(* Logix 5000 project; controller MetsoFilter vendor 1 type 14 code 106 rev 32.11; software revision 32.00; part 2 of 4 *)
(* tags used below, declared in another part *)
   AlarmReset : BOOL;   // Alarm Rest Relay
   ALM_AirAndWaterOK_T : TIMER;   // Air and Water OK, Enable Air & Water Valves Alarms
   ALM_W1 : DINT;   // Alarms to HMI, Word #1
   ALM_W2 : DINT;   // Alarms to HMI, Word #2
   AS_AirDry : BOOL;   // Auto Sequence, Air Dry
   AS_ClothFlush : BOOL;   // Auto Sequence Flush out Cloth
   AS_ClothFlush_T : TIMER;   // Auto Sequence Flush out Cloth Timer
   AS_ClothVibWash : BOOL;   // Auto Sequence Vibrate & Wash Cloth
   AS_ClothVibWash_T : TIMER;   // Auto Sequence Vibrate & Wash Cloth Timer
   AS_Done : BOOL;   // Automatic Sequence Done, Reset Sequence for Next Run
   AS_Drain : BOOL;   // Auto Sequence, Drain
   AS_FeedFilter : BOOL;   // Auto Sequence, Feed Filter
   AS_HighEmptyWeight : BOOL;   // Auto Sequence, High Empty Weight, Manually Shake filter
   AS_HighPressClose : BOOL;   // Auto Sequence, Close Press at High Pressure
   AS_LowFeedWeight : BOOL;   // Auto Sequence, Low Feed Weight, Enable Retry
   AS_LowPressClose : BOOL;   // Auto Sequence, Close Press at Low Pressure
   AS_MembComp : BOOL;   // Auto Sequence, Membrane Compress
   AS_TopBlowAir1 : BOOL;   // Auto Sequence, Top Blow Air #1
   AS_TopBlowAir2 : BOOL;   // Auto Sequence, Top Blow Air #2
   AS_TopBlowWat : BOOL;   // Automatic Sequence, Top Blow & Water
   AS_VibrateCloth : BOOL;   // Auto Sequence Vibrate Cloth
   AS_VibrateCloth_T : TIMER;   // Auto Sequence Vibrate Cloth Timer
   AS_Wait : BOOL;   // Auto Sequence Wait
   AS_Wait_T : TIMER;   // Auto Sequence Wait Timer
   At_Parked_Pos_T : TIMER;   // Press At Parked (Closed) Postion Timer
   Auto_ON : BOOL;   // Auto On Mode
   Auto_Run : BOOL;   // Run the Next Step of the Auto Sequence
   AutoSeqStarted : BOOL;   // Auto Sequence Started
   DD_PressPressure : REAL;   // Press Pressure Data Display
   DD_PressWeight : DINT;   // Press Weight from Analog Input Data Display
   DE_ClothVibWash : DINT;   // Settings Screen, Cloth Vibrate and Wash Time Data Entry (Seconds)
   DE_ClothWash : DINT;   // Settings Screen, Cloth Wash Time Data Entry (Seconds)
   DE_DelayedStart : DINT;   // Settings Screen, Delay Start Wait Time Data Entry (Seconds)
   DryAirSwitch : BOOL;   // Drying Air OK Switch
   Goto_Neutral_T : TIMER;   // Manual / Auto Open (Goto Neutral) Press On Plus Time
   Goto_Park_T : TIMER;   // Go to Park On Plus Time
   Goto_Press_T : TIMER;   // Go to Press Position Output On Plus Time
   GS3 : BOOL;   // Press At Park Position Prox Switch
   GS4 : BOOL;   // Press At Neutral Position Prox Switch
   GS8 : BOOL;   // Press At Press Position Prox Switch
   GSC11 : BOOL;   // Upper Hatch is Closed Proximity Switch
   GSC9 : BOOL;   // Lower Hatch is Closed Proximity Switch
   GSO10 : BOOL;   // Lower Hatch is Open Proximity Switch
   GSO12 : BOOL;   // Upper Hatch is Open Proximity Switch
   H4a : BOOL;   // Hydraulic Valve, Raise (Open) Lower Hatch
   H4a_On_T : TIMER;   // Hydraulic Valve, Raise (Open) Lower Hatch On Plus Time
   H4b : BOOL;   // Hydraulic Valve, Lower (Close) Lower Hatch
   H4b_On_T : TIMER;   // Hydraulic Valve, Lower (Close) Lower Hatch On Plus Time
   H5a : BOOL;   // Hydraulic Valve, Raise (Open) Upper Hatch
   H5a_On_T : TIMER;   // Hydraulic Valve, Raise (Open) Upper Hatch On Plus Time
   H5b : BOOL;   // Hydraulic Valve, Lower (Close) Upper Hatch
   H5b_On_T : TIMER;   // Hydraulic Valve, Lower (Close) Upper Hatch On Plus Time
   HPP_Run_T : TIMER;   // High Pressure Pump Run Timer
   LPP_Run_T : TIMER;   // Low Pressure Pump Run Timer
   M_HPP_Run : BOOL;   // High Pressure Pump Run Output Bit
   M_HPP_Running : BOOL;   // High Pressure Pump is Running
   M_LPP_Run : BOOL;   // Low Pressure Pump Run Output Bit
   M_LPP_Running : BOOL;   // Low Pressure Pump is Running
   MAN_ClosePress : BOOL;   // Manual Close Press to Park Position
   Manual_ON : BOOL;   // Manual On Mode
   MAS_CloseHatch : BOOL;   // Manual / Auto Close Hatch
   MAS_HatchesClosed_T : TIMER;   // Manual / Auto Hatchs are Closed + Time
   MAS_OpenHatch : BOOL;   // Manual / Auto Open Hatch
   MAS_OpenPress : BOOL;   // Manual / Auto Open (Goto Neutral) Press
   MSG_Activity : DINT;   // Activity Message display at left side of the HMI Screens.
   MSG_CloseHatch : BOOL;   // Show Closing Hatches in Sequence & Activity messages latch
   MSG_Main : DINT;   // Main Message at center of screen,
   MSG_MainTemp : DINT;   // Main Message at center of screen, Temporary Holding Register
   MSG_OpenHatch : BOOL;   // Show Opeining Hatch in SEquence & Activity messages latch
   MSG_OpenPress : BOOL;   // Show Opeining Press in Sequence & Activity messages latch
   MSG_SeqTemp : DINT;   // Sequence & Activity Message displays at left side of the HMI Screens, Temp hold
   MSG_Sequence : DINT;   // Sequence Message display at left side of the HMI Screens.
   NumberOfAlarms : DINT;   // Number of Active Alarms
   PressPressure_OOR_T : TIMER;   // Press Pressure Sensor Out Of Range Plus Time
   PressWeight_OOR_T : TIMER;   // Press Weight Out Of Range Timer
   SlurrySystemSwitch : BOOL;   // Slurry System OK Switch
   V10_GSC : BOOL;   // Valve #10, Membrane Drain, Closed Input
   V10_Off_T : TIMER;   // Valve #10, Membrane Drain, Ouput Bit Off Plus Time, Valve shoud be Open
   V10_On_T : TIMER;   // Valve #10, Membrane Drain, Ouput Bit On Plus Time, Valve shoud be Closed
   V1_GSC : BOOL;   // Valve #1, Slurry Supply, Closed Input
   V1_GSO : BOOL;   // Valve #1, Slurry Supply, Open Input
   V1_Off_T : TIMER;   // Valve #1, Slurry Supply, Open Output Bit Off Plus Time
   V1_On_T : TIMER;   // Valve #1, Slurry Supply, Open Output Bit On Plus Time
   V3_GSC : BOOL;   // Valve #3, Filtrate, Closed Input
   V3_GSO : BOOL;   // Valve #3, Filtrate, Open Input
   V3_Off_T : TIMER;   // Valve #3, Filtrate, Open Output Bit Off Plus time
   V3_On_T : TIMER;   // Valve #3, Filtrate, Open Output Bit On Plus time
   V4_GSC : BOOL;   // Valve #4, Slurry Return, Closed Input
   V4_GSO : BOOL;   // Valve #4, Slurry Return, Open Input
   V4_Off_T : TIMER;   // Valve #4, Slurry Return, Open Output Bit Off Plus Time
   V4_On_T : TIMER;   // Valve #4, Slurry Return, Open Output Bit On Plus Time
   V5_GSC : BOOL;   // Valve #5, Drying Air, Closed Input
   V5_GSO : BOOL;   // Valve #5, Drying Air, Opened Input
   V5_Off_T : TIMER;   // Valve #5, Drying Air, Open Output Bit Off Plus Time
   V5_On_T : TIMER;   // Valve #5, Drying Air, Open Output Bit On Plus Time
   V6_GSC : BOOL;   // Valve #6, Top Blow Air, Closed Input
   V6_GSO : BOOL;   // Valve #6, Top Blow Air, Opened Input
   V6_Off_T : TIMER;   // Valve #6, Top Blow Air, Open Output Bit On Plus Time
   V6_On_T : TIMER;   // Valve #6, Top Blow Air, Open Output Bit On Plus Time
   V7_GSC : BOOL;   // Valve #7, Membrane Air, Closed Input
   V7_GSO : BOOL;   // Valve #7, Membrane Air, Opened Input
   V7_Off_T : TIMER;   // Valve #7, Membrane Air, Open Output Bit Off Plus Time
   V7_On_T : TIMER;   // Valve #7, Membrane Air, Open Output Bit On Plus time
   V8_GSC : BOOL;   // Valve #8, Top Blow Water, Closed Input
   V8_GSO : BOOL;   // Valve #8, Top Blow Water, Opened Input
   V8_Off_T : TIMER;   // Valve #8, Top Blow Water, Open Output Bit Off Plus Time
   V8_On_T : TIMER;   // Valve #8, Top Blow Water, Open Output Bit On Plus Time
   V9_GSC : BOOL;   // Valve #9, Wash Water, Closed Input
   V9_GSO : BOOL;   // Valve #9, Wash Water, Opened Input
   V9_Off_T : TIMER;   // Valve #9, Wash Water, Open Ouput Bit Off Plus Time
   V9_On_T : TIMER;   // Valve #9, Wash Water, Open Ouput Bit On Plus Time
   WashWaterSwitch : BOOL;   // Wash Water System OK Switch
   YV1 : BOOL;   // Valve #1, Slurry Supply, Open Output Bit
   YV10 : BOOL;   // Valve #10, Membrane Drain, Normally Open, Energize to Close, Output Bit
   YV3 : BOOL;   // Valve #3, Filtrate, Open Output Bit
   YV4 : BOOL;   // Valve #4, Slurry Return, Open Output Bit
   YV5 : BOOL;   // Valve #5, Drying Air, Open Output Bit
   YV6 : BOOL;   // Valve #6, Top Blow Air, Open Output Bit
   YV7 : BOOL;   // Valve #7, Membrane Air, Open Output Bit
   YV8 : BOOL;   // Valve #8, Top Blow Water, Open Output Bit
   YV9 : BOOL;   // Valve #9, Wash Water, Open Ouput Bit
(* MainProgram, continued *)

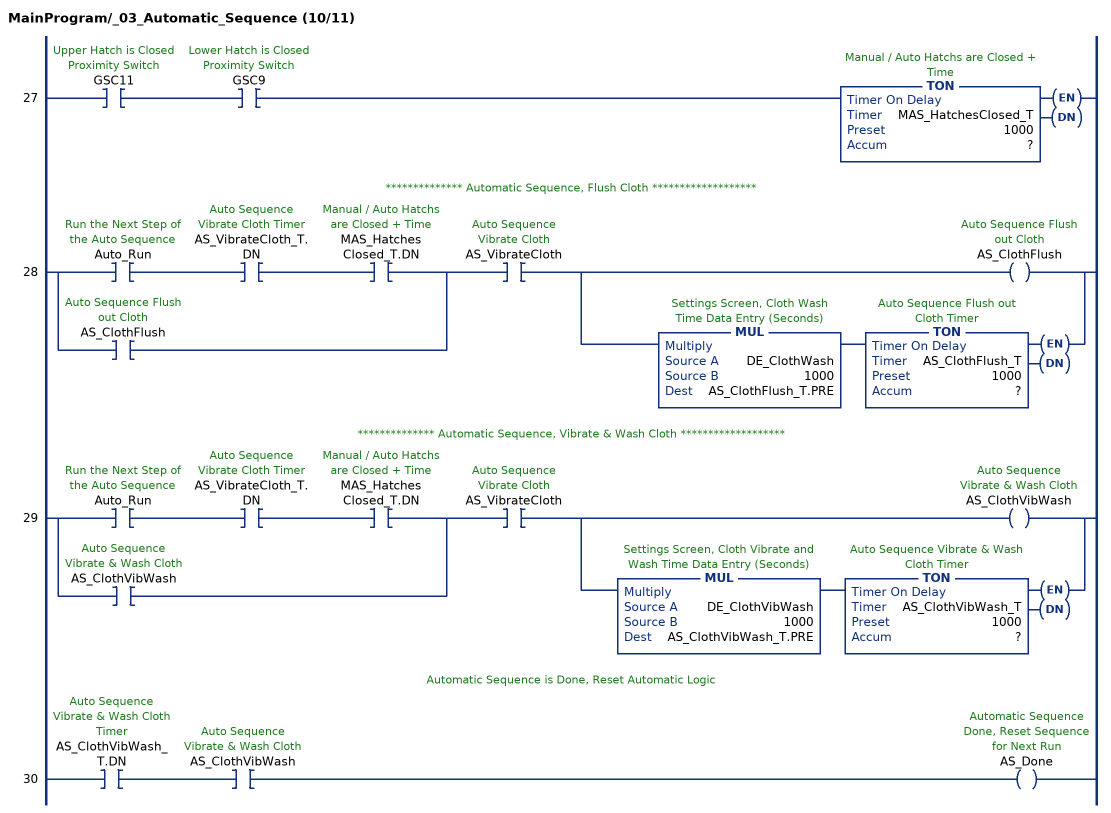
   [picture p24: MainProgram/_03_Automatic_Sequence rungs 27-30]
   27: XIC(GSC11)XIC(GSC9)TON(MAS_HatchesClosed_T,?,?);
   // ************** Automatic Sequence, Flush Cloth *******************
   28: [XIC(Auto_Run) XIC(AS_VibrateCloth_T.DN) XIC(MAS_HatchesClosed_T.DN) ,XIC(AS_ClothFlush) ]XIC(AS_VibrateCloth)[OTE(AS_ClothFlush) ,MUL(DE_ClothWash,1000,AS_ClothFlush_T.PRE) TON(AS_ClothFlush_T,?,?) ];
   // ************** Automatic Sequence, Vibrate & Wash Cloth *******************
   29: [XIC(Auto_Run) XIC(AS_VibrateCloth_T.DN) XIC(MAS_HatchesClosed_T.DN) ,XIC(AS_ClothVibWash) ]XIC(AS_VibrateCloth)[OTE(AS_ClothVibWash) ,MUL(DE_ClothVibWash,1000,AS_ClothVibWash_T.PRE) TON(AS_ClothVibWash_T,?,?) ];
   // Automatic Sequence is Done, Reset Automatic Logic
   30: XIC(AS_ClothVibWash_T.DN)XIC(AS_ClothVibWash)OTE(AS_Done);
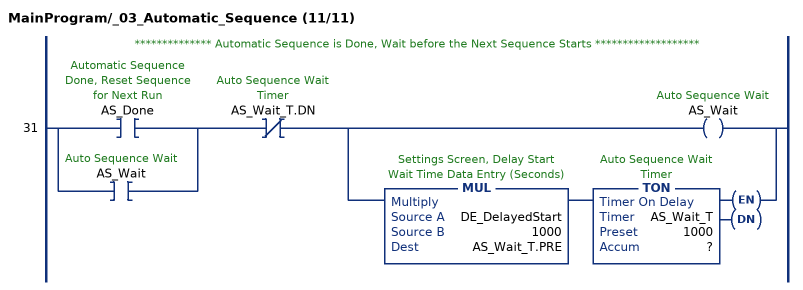
   // ************** Automatic Sequence is Done, Wait before the Next Sequence Starts *******************
   31: [XIC(AS_Done) ,XIC(AS_Wait) ]XIO(AS_Wait_T.DN)[OTE(AS_Wait) ,MUL(DE_DelayedStart,1000,AS_Wait_T.PRE) TON(AS_Wait_T,?,?) ];
END_ROUTINE

ROUTINE _04_HMI_MessageDisplays   (* ladder *)
// Message Displays on HMI Screens
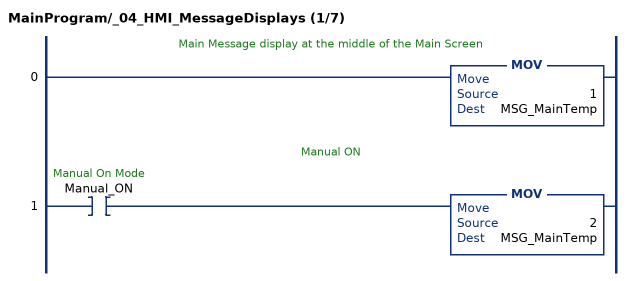
   // Main Message display at the middle of the Main Screen
   0: MOV(1,MSG_MainTemp);
   // Manual ON
   1: XIC(Manual_ON)MOV(2,MSG_MainTemp);
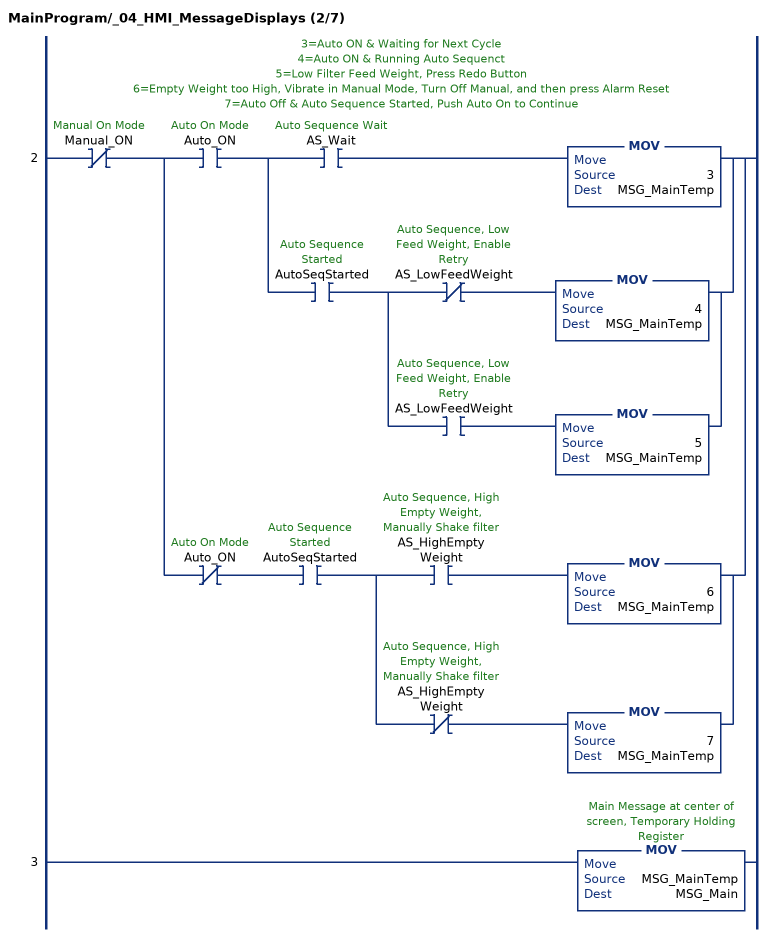
   // 3=Auto ON & Waiting for Next Cycle
   // 4=Auto ON & Running Auto Sequenct
   // 5=Low Filter Feed Weight, Press Redo Button
   // 6=Empty Weight too High, Vibrate in Manual Mode, Turn Off Manual, and then press Alarm Reset
   // 7=Auto Off & Auto Sequence Started, Push Auto On to Continue
   2: XIO(Manual_ON)[XIC(Auto_ON) [XIC(AS_Wait) MOV(3,MSG_MainTemp) ,XIC(AutoSeqStarted) [XIO(AS_LowFeedWeight) MOV(4,MSG_MainTemp) ,XIC(AS_LowFeedWeight) MOV(5,MSG_MainTemp) ] ] ,XIO(Auto_ON) XIC(AutoSeqStarted) [XIC(AS_HighEmptyWeight) MOV(6,MSG_MainTemp) ,XIO(AS_HighEmptyWeight) MOV(7,MSG_MainTemp) ] ];
   3: MOV(MSG_MainTemp,MSG_Main);
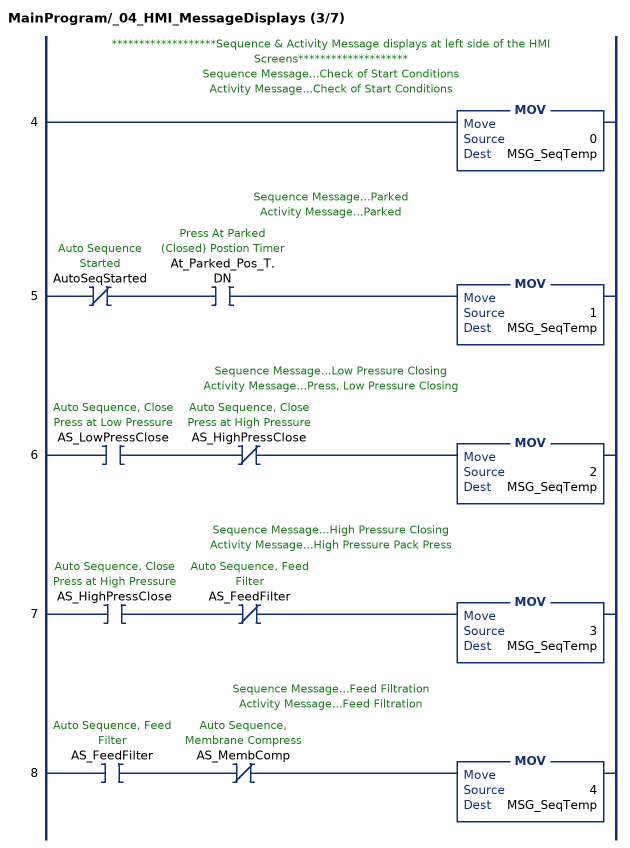
   // *******************Sequence & Activity Message displays at left side of the HMI Screens********************
   // Sequence Message...Check of Start Conditions
   // Activity Message...Check of Start Conditions
   4: MOV(0,MSG_SeqTemp);
   // Sequence Message...Parked
   // Activity Message...Parked
   5: XIO(AutoSeqStarted)XIC(At_Parked_Pos_T.DN)MOV(1,MSG_SeqTemp);
   // Sequence Message...Low Pressure Closing
   // Activity Message...Press, Low Pressure Closing
   6: XIC(AS_LowPressClose)XIO(AS_HighPressClose)MOV(2,MSG_SeqTemp);
   // Sequence Message...High Pressure Closing
   // Activity Message...High Pressure Pack Press
   7: XIC(AS_HighPressClose)XIO(AS_FeedFilter)MOV(3,MSG_SeqTemp);
   // Sequence Message...Feed Filtration
   // Activity Message...Feed Filtration
   8: XIC(AS_FeedFilter)XIO(AS_MembComp)MOV(4,MSG_SeqTemp);
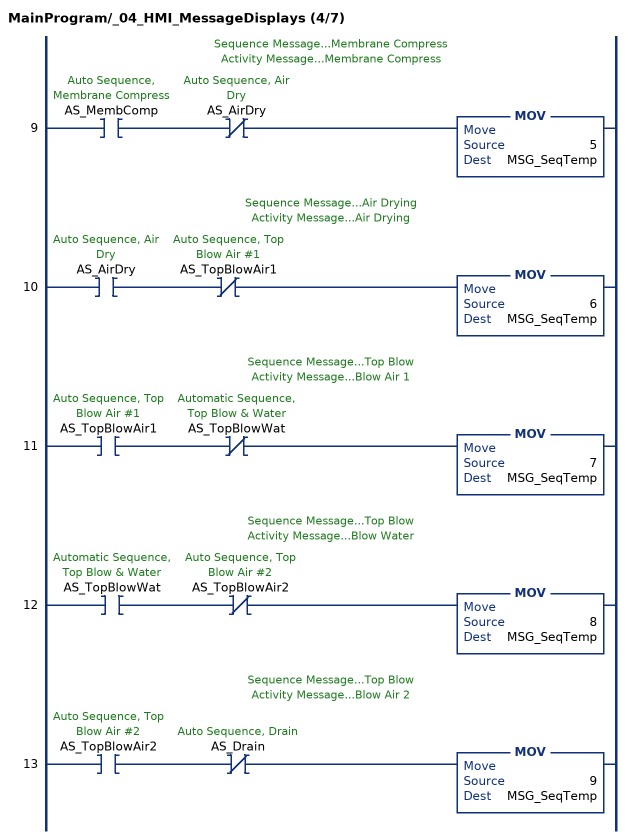
   // Sequence Message...Membrane Compress
   // Activity Message...Membrane Compress
   9: XIC(AS_MembComp)XIO(AS_AirDry)MOV(5,MSG_SeqTemp);
   // Sequence Message...Air Drying
   // Activity Message...Air Drying
   10: XIC(AS_AirDry)XIO(AS_TopBlowAir1)MOV(6,MSG_SeqTemp);
   // Sequence Message...Top Blow
   // Activity Message...Blow Air 1
   11: XIC(AS_TopBlowAir1)XIO(AS_TopBlowWat)MOV(7,MSG_SeqTemp);
   // Sequence Message...Top Blow
   // Activity Message...Blow Water
   12: XIC(AS_TopBlowWat)XIO(AS_TopBlowAir2)MOV(8,MSG_SeqTemp);
   // Sequence Message...Top Blow
   // Activity Message...Blow Air 2
   13: XIC(AS_TopBlowAir2)XIO(AS_Drain)MOV(9,MSG_SeqTemp);
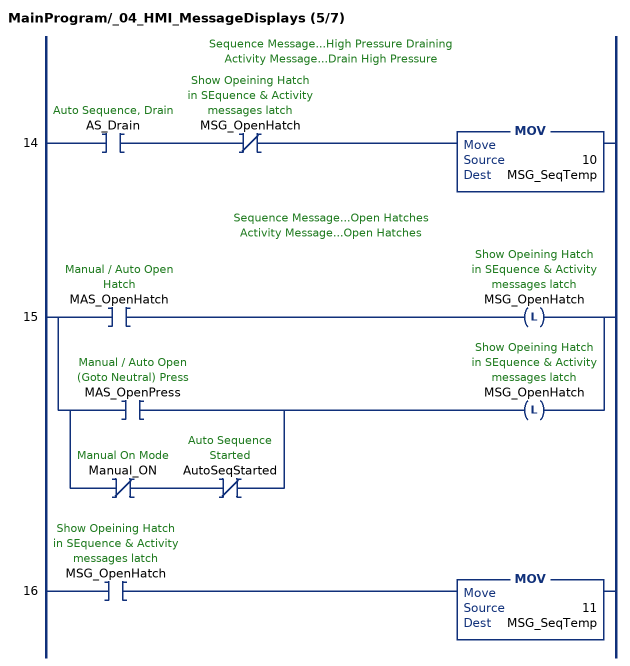
   // Sequence Message...High Pressure Draining
   // Activity Message...Drain High Pressure
   14: XIC(AS_Drain)XIO(MSG_OpenHatch)MOV(10,MSG_SeqTemp);
   // Sequence Message...Open Hatches
   // Activity Message...Open Hatches
   15: [XIC(MAS_OpenHatch) OTL(MSG_OpenHatch) ,[XIC(MAS_OpenPress) ,XIO(Manual_ON) XIO(AutoSeqStarted) ] OTL(MSG_OpenHatch) ];
   16: XIC(MSG_OpenHatch)MOV(11,MSG_SeqTemp);
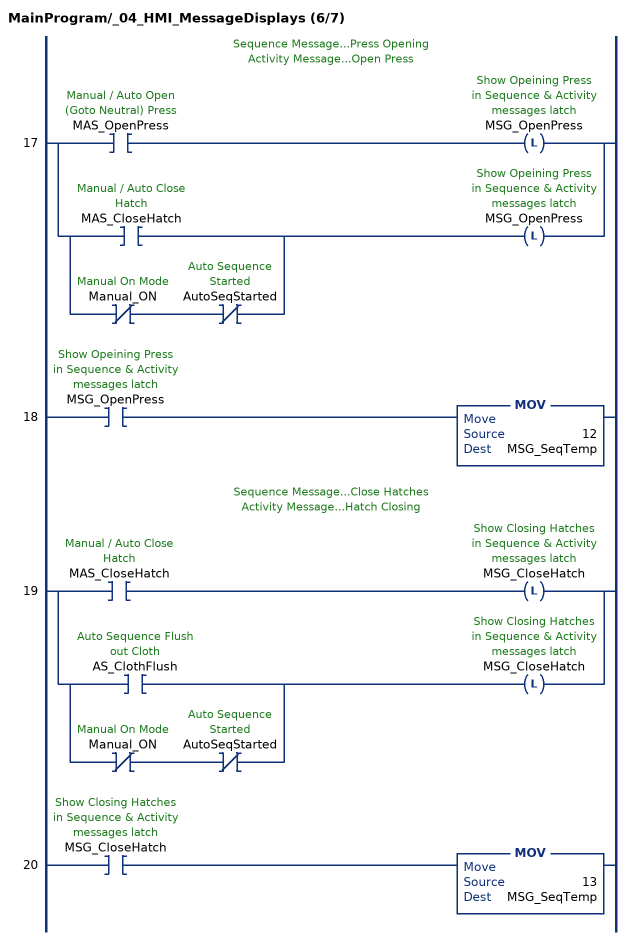
   // Sequence Message...Press Opening
   // Activity Message...Open Press
   17: [XIC(MAS_OpenPress) OTL(MSG_OpenPress) ,[XIC(MAS_CloseHatch) ,XIO(Manual_ON) XIO(AutoSeqStarted) ] OTL(MSG_OpenPress) ];
   18: XIC(MSG_OpenPress)MOV(12,MSG_SeqTemp);
   // Sequence Message...Close Hatches
   // Activity Message...Hatch Closing
   19: [XIC(MAS_CloseHatch) OTL(MSG_CloseHatch) ,[XIC(AS_ClothFlush) ,XIO(Manual_ON) XIO(AutoSeqStarted) ] OTL(MSG_CloseHatch) ];
   20: XIC(MSG_CloseHatch)MOV(13,MSG_SeqTemp);
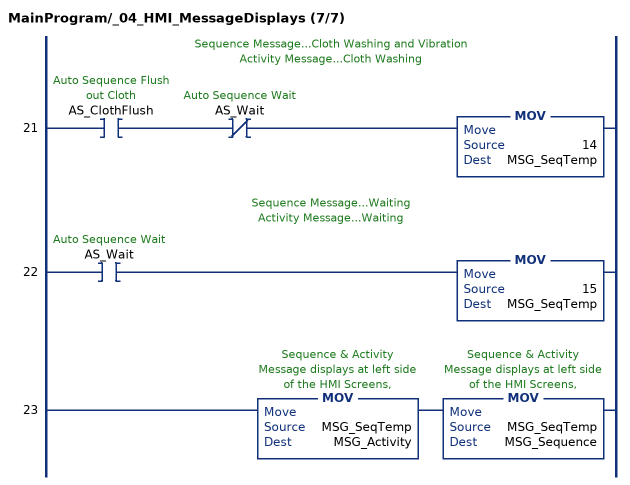
   // Sequence Message...Cloth Washing and Vibration
   // Activity Message...Cloth Washing
   21: XIC(AS_ClothFlush)XIO(AS_Wait)MOV(14,MSG_SeqTemp);
   // Sequence Message...Waiting
   // Activity Message...Waiting
   22: XIC(AS_Wait)MOV(15,MSG_SeqTemp);
   23: MOV(MSG_SeqTemp,MSG_Activity)MOV(MSG_SeqTemp,MSG_Sequence);
END_ROUTINE

ROUTINE _05_Alarms   (* ladder *)
// Alarms Logic
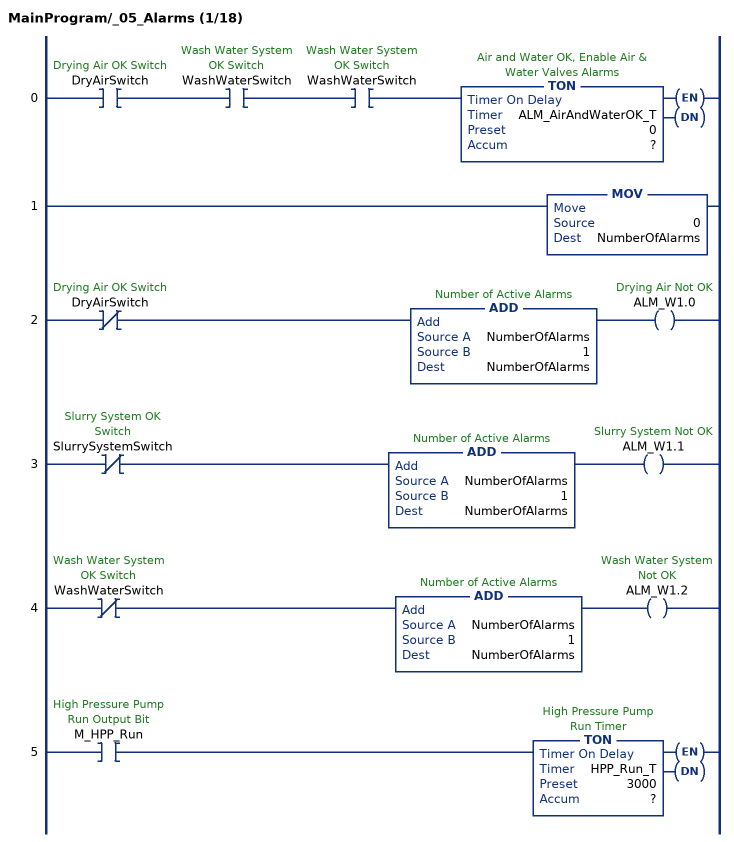
   0: XIC(DryAirSwitch)XIC(WashWaterSwitch)XIC(WashWaterSwitch)TON(ALM_AirAndWaterOK_T,?,?);
   1: MOV(0,NumberOfAlarms);
   2: XIO(DryAirSwitch)ADD(NumberOfAlarms,1,NumberOfAlarms)OTE(ALM_W1.0);
   3: XIO(SlurrySystemSwitch)ADD(NumberOfAlarms,1,NumberOfAlarms)OTE(ALM_W1.1);
   4: XIO(WashWaterSwitch)ADD(NumberOfAlarms,1,NumberOfAlarms)OTE(ALM_W1.2);
   5: XIC(M_HPP_Run)TON(HPP_Run_T,?,?);
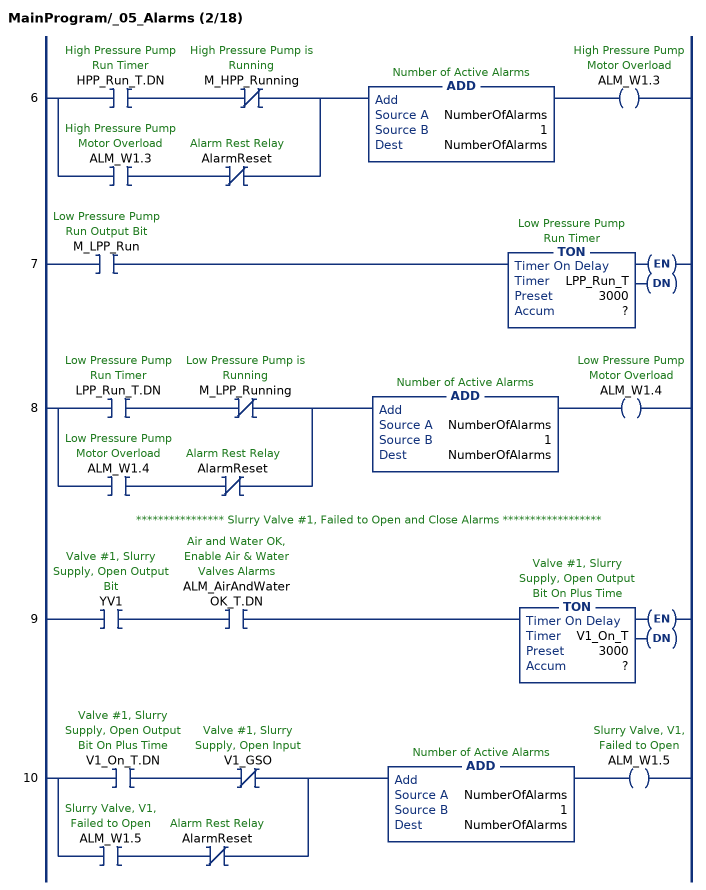
   6: [XIC(HPP_Run_T.DN) XIO(M_HPP_Running) ,XIC(ALM_W1.3) XIO(AlarmReset) ]ADD(NumberOfAlarms,1,NumberOfAlarms)OTE(ALM_W1.3);
   7: XIC(M_LPP_Run)TON(LPP_Run_T,?,?);
   8: [XIC(LPP_Run_T.DN) XIO(M_LPP_Running) ,XIC(ALM_W1.4) XIO(AlarmReset) ]ADD(NumberOfAlarms,1,NumberOfAlarms)OTE(ALM_W1.4);
   // **************** Slurry Valve #1, Failed to Open and Close Alarms ******************
   9: XIC(YV1)XIC(ALM_AirAndWaterOK_T.DN)TON(V1_On_T,?,?);
   10: [XIC(V1_On_T.DN) XIO(V1_GSO) ,XIC(ALM_W1.5) XIO(AlarmReset) ]ADD(NumberOfAlarms,1,NumberOfAlarms)OTE(ALM_W1.5);
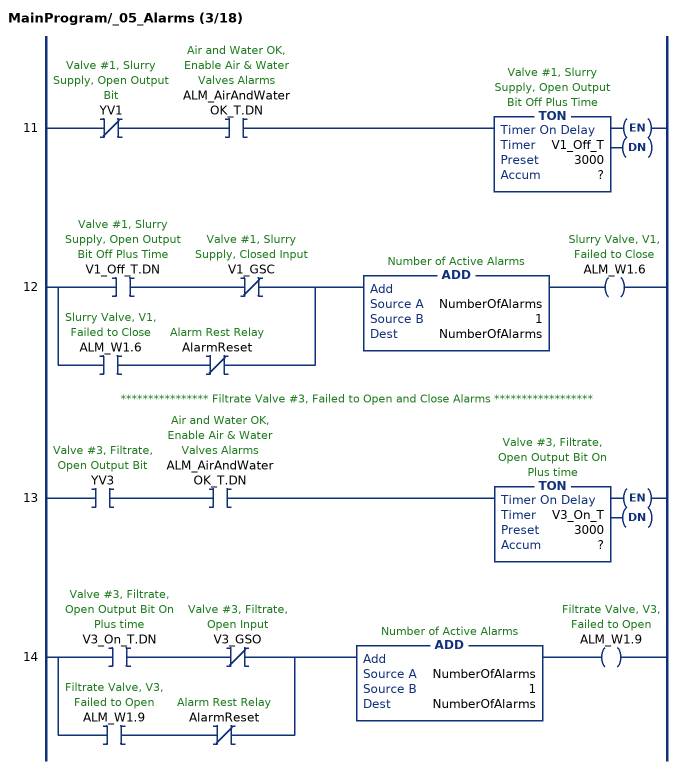
   11: XIO(YV1)XIC(ALM_AirAndWaterOK_T.DN)TON(V1_Off_T,?,?);
   12: [XIC(V1_Off_T.DN) XIO(V1_GSC) ,XIC(ALM_W1.6) XIO(AlarmReset) ]ADD(NumberOfAlarms,1,NumberOfAlarms)OTE(ALM_W1.6);
   // **************** Filtrate Valve #3, Failed to Open and Close Alarms ******************
   13: XIC(YV3)XIC(ALM_AirAndWaterOK_T.DN)TON(V3_On_T,?,?);
   14: [XIC(V3_On_T.DN) XIO(V3_GSO) ,XIC(ALM_W1.9) XIO(AlarmReset) ]ADD(NumberOfAlarms,1,NumberOfAlarms)OTE(ALM_W1.9);
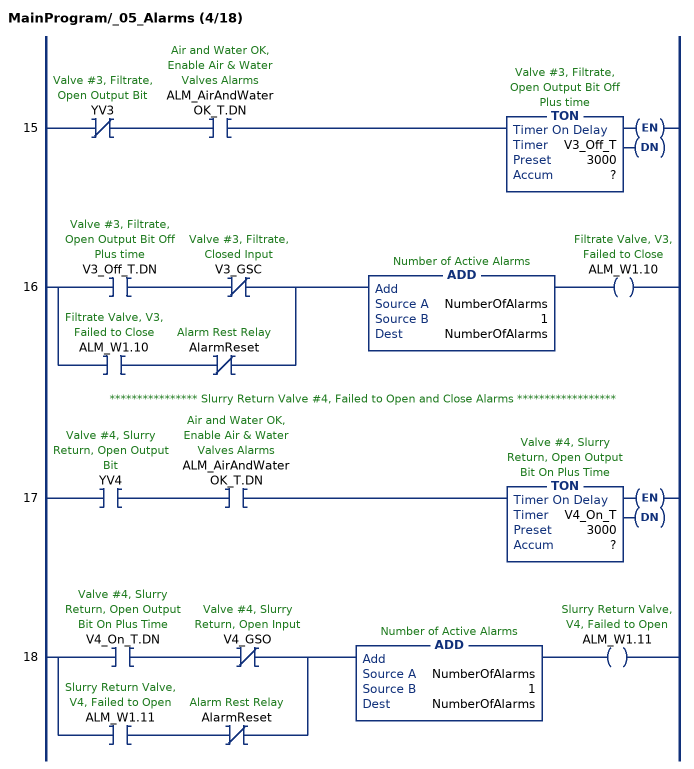
   15: XIO(YV3)XIC(ALM_AirAndWaterOK_T.DN)TON(V3_Off_T,?,?);
   16: [XIC(V3_Off_T.DN) XIO(V3_GSC) ,XIC(ALM_W1.10) XIO(AlarmReset) ]ADD(NumberOfAlarms,1,NumberOfAlarms)OTE(ALM_W1.10);
   // **************** Slurry Return Valve #4, Failed to Open and Close Alarms ******************
   17: XIC(YV4)XIC(ALM_AirAndWaterOK_T.DN)TON(V4_On_T,?,?);
   18: [XIC(V4_On_T.DN) XIO(V4_GSO) ,XIC(ALM_W1.11) XIO(AlarmReset) ]ADD(NumberOfAlarms,1,NumberOfAlarms)OTE(ALM_W1.11);
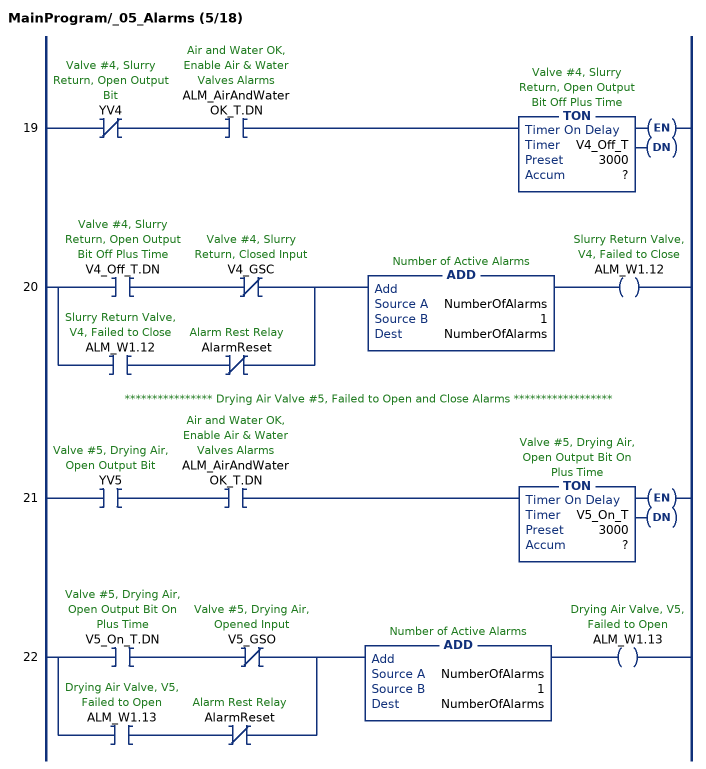
   19: XIO(YV4)XIC(ALM_AirAndWaterOK_T.DN)TON(V4_Off_T,?,?);
   20: [XIC(V4_Off_T.DN) XIO(V4_GSC) ,XIC(ALM_W1.12) XIO(AlarmReset) ]ADD(NumberOfAlarms,1,NumberOfAlarms)OTE(ALM_W1.12);
   // **************** Drying Air Valve #5, Failed to Open and Close Alarms ******************
   21: XIC(YV5)XIC(ALM_AirAndWaterOK_T.DN)TON(V5_On_T,?,?);
   22: [XIC(V5_On_T.DN) XIO(V5_GSO) ,XIC(ALM_W1.13) XIO(AlarmReset) ]ADD(NumberOfAlarms,1,NumberOfAlarms)OTE(ALM_W1.13);
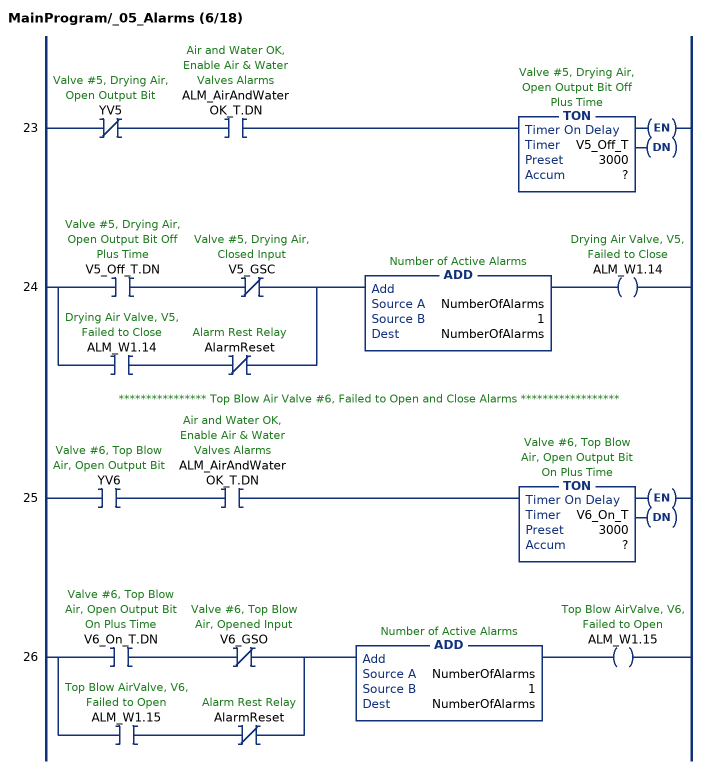
   23: XIO(YV5)XIC(ALM_AirAndWaterOK_T.DN)TON(V5_Off_T,?,?);
   24: [XIC(V5_Off_T.DN) XIO(V5_GSC) ,XIC(ALM_W1.14) XIO(AlarmReset) ]ADD(NumberOfAlarms,1,NumberOfAlarms)OTE(ALM_W1.14);
   // **************** Top Blow Air Valve #6, Failed to Open and Close Alarms ******************
   25: XIC(YV6)XIC(ALM_AirAndWaterOK_T.DN)TON(V6_On_T,?,?);
   26: [XIC(V6_On_T.DN) XIO(V6_GSO) ,XIC(ALM_W1.15) XIO(AlarmReset) ]ADD(NumberOfAlarms,1,NumberOfAlarms)OTE(ALM_W1.15);
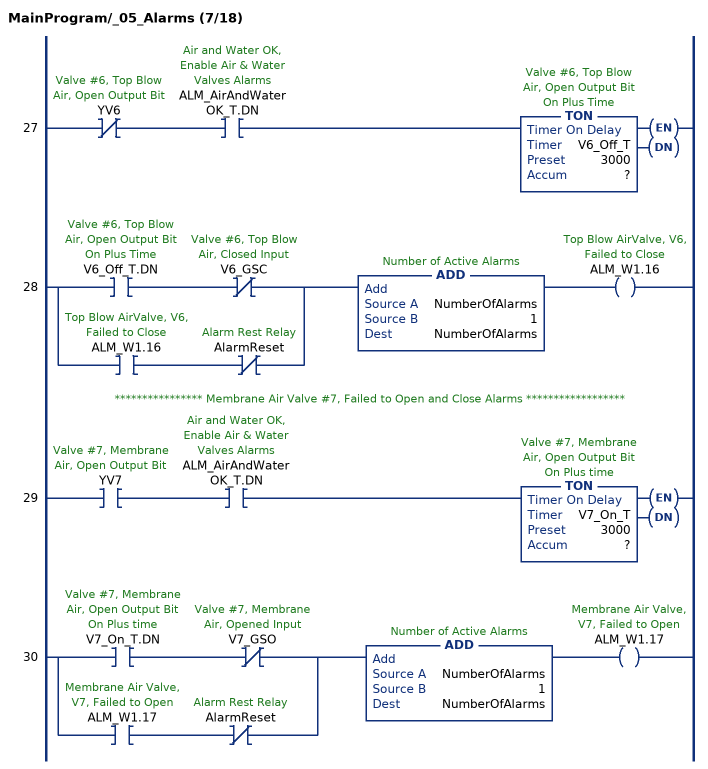
   27: XIO(YV6)XIC(ALM_AirAndWaterOK_T.DN)TON(V6_Off_T,?,?);
   28: [XIC(V6_Off_T.DN) XIO(V6_GSC) ,XIC(ALM_W1.16) XIO(AlarmReset) ]ADD(NumberOfAlarms,1,NumberOfAlarms)OTE(ALM_W1.16);
   // **************** Membrane Air Valve #7, Failed to Open and Close Alarms ******************
   29: XIC(YV7)XIC(ALM_AirAndWaterOK_T.DN)TON(V7_On_T,?,?);
   30: [XIC(V7_On_T.DN) XIO(V7_GSO) ,XIC(ALM_W1.17) XIO(AlarmReset) ]ADD(NumberOfAlarms,1,NumberOfAlarms)OTE(ALM_W1.17);
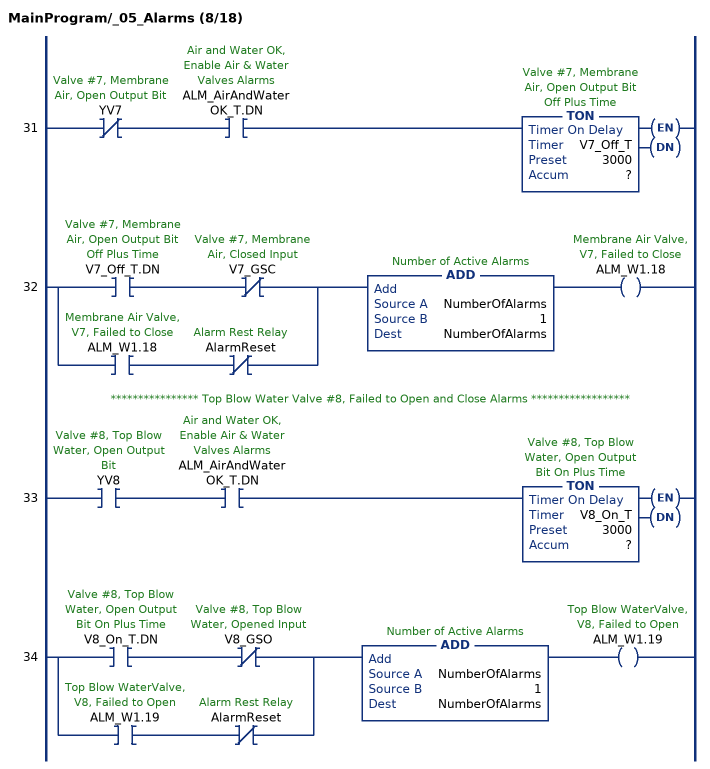
   31: XIO(YV7)XIC(ALM_AirAndWaterOK_T.DN)TON(V7_Off_T,?,?);
   32: [XIC(V7_Off_T.DN) XIO(V7_GSC) ,XIC(ALM_W1.18) XIO(AlarmReset) ]ADD(NumberOfAlarms,1,NumberOfAlarms)OTE(ALM_W1.18);
   // **************** Top Blow Water Valve #8, Failed to Open and Close Alarms ******************
   33: XIC(YV8)XIC(ALM_AirAndWaterOK_T.DN)TON(V8_On_T,?,?);
   34: [XIC(V8_On_T.DN) XIO(V8_GSO) ,XIC(ALM_W1.19) XIO(AlarmReset) ]ADD(NumberOfAlarms,1,NumberOfAlarms)OTE(ALM_W1.19);
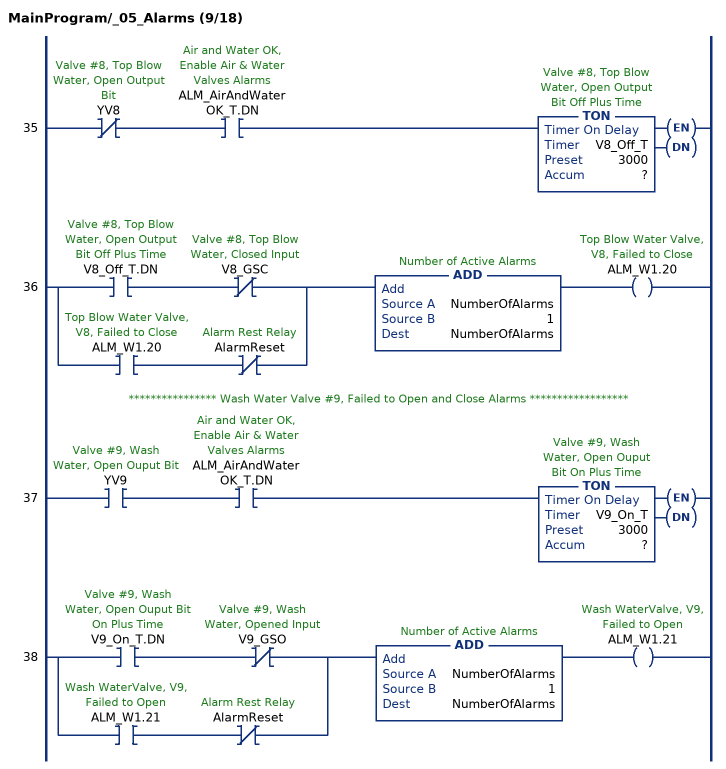
   35: XIO(YV8)XIC(ALM_AirAndWaterOK_T.DN)TON(V8_Off_T,?,?);
   36: [XIC(V8_Off_T.DN) XIO(V8_GSC) ,XIC(ALM_W1.20) XIO(AlarmReset) ]ADD(NumberOfAlarms,1,NumberOfAlarms)OTE(ALM_W1.20);
   // **************** Wash Water Valve #9, Failed to Open and Close Alarms ******************
   37: XIC(YV9)XIC(ALM_AirAndWaterOK_T.DN)TON(V9_On_T,?,?);
   38: [XIC(V9_On_T.DN) XIO(V9_GSO) ,XIC(ALM_W1.21) XIO(AlarmReset) ]ADD(NumberOfAlarms,1,NumberOfAlarms)OTE(ALM_W1.21);
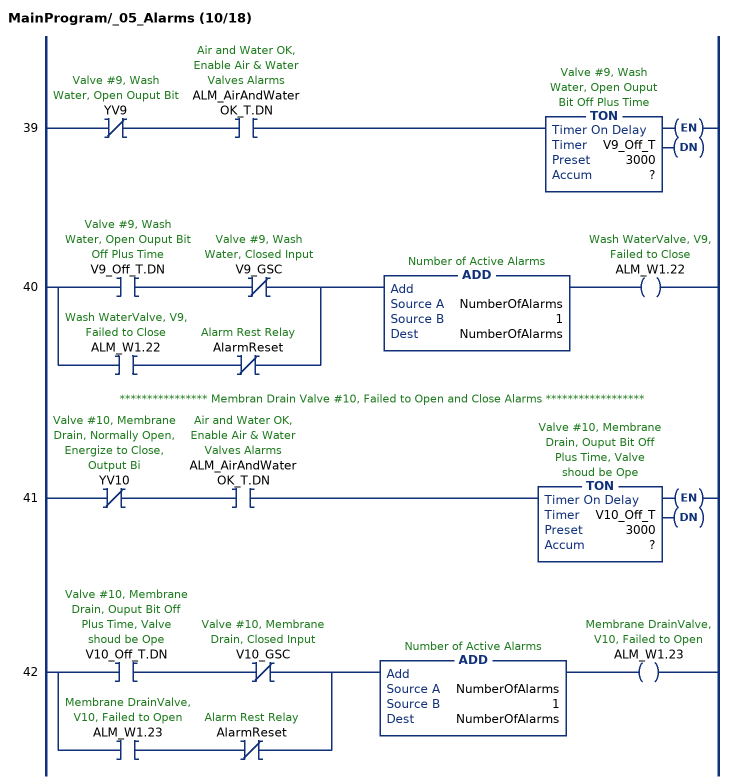
   39: XIO(YV9)XIC(ALM_AirAndWaterOK_T.DN)TON(V9_Off_T,?,?);
   40: [XIC(V9_Off_T.DN) XIO(V9_GSC) ,XIC(ALM_W1.22) XIO(AlarmReset) ]ADD(NumberOfAlarms,1,NumberOfAlarms)OTE(ALM_W1.22);
   // **************** Membran Drain Valve #10, Failed to Open and Close Alarms ******************
   41: XIO(YV10)XIC(ALM_AirAndWaterOK_T.DN)TON(V10_Off_T,?,?);
   42: [XIC(V10_Off_T.DN) XIO(V10_GSC) ,XIC(ALM_W1.23) XIO(AlarmReset) ]ADD(NumberOfAlarms,1,NumberOfAlarms)OTE(ALM_W1.23);
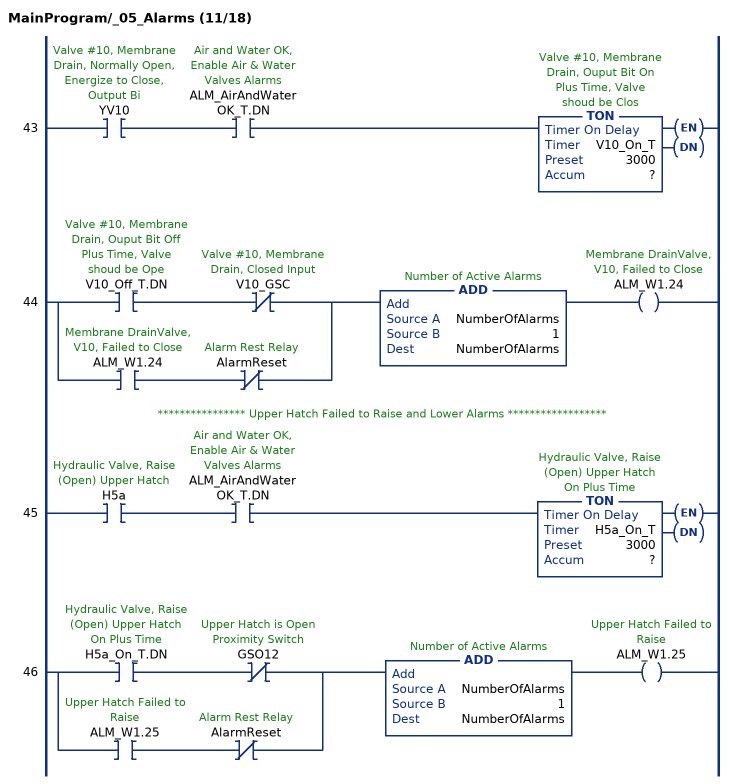
   43: XIC(YV10)XIC(ALM_AirAndWaterOK_T.DN)TON(V10_On_T,?,?);
   44: [XIC(V10_Off_T.DN) XIO(V10_GSC) ,XIC(ALM_W1.24) XIO(AlarmReset) ]ADD(NumberOfAlarms,1,NumberOfAlarms)OTE(ALM_W1.24);
   // **************** Upper Hatch Failed to Raise and Lower Alarms ******************
   45: XIC(H5a)XIC(ALM_AirAndWaterOK_T.DN)TON(H5a_On_T,?,?);
   46: [XIC(H5a_On_T.DN) XIO(GSO12) ,XIC(ALM_W1.25) XIO(AlarmReset) ]ADD(NumberOfAlarms,1,NumberOfAlarms)OTE(ALM_W1.25);
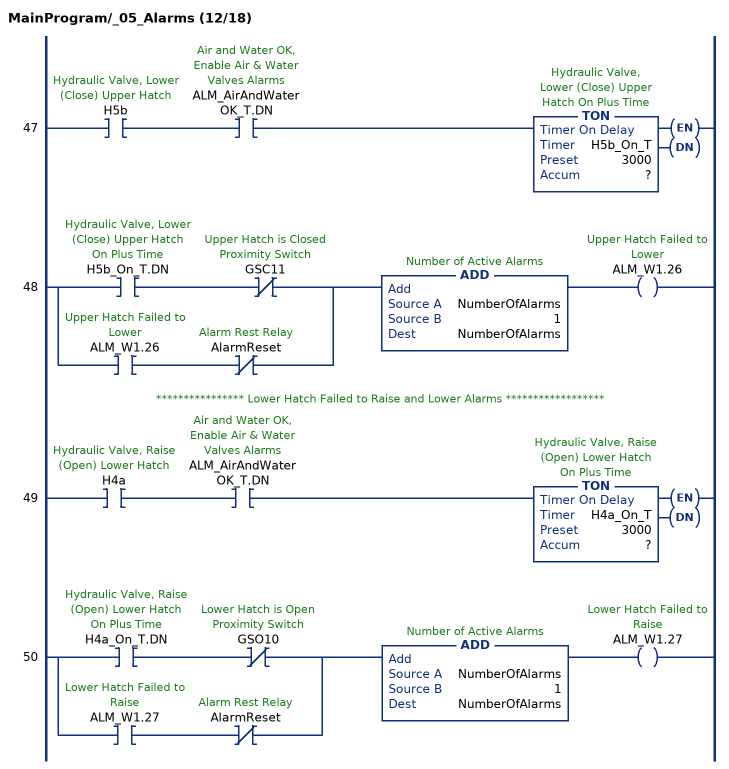
   47: XIC(H5b)XIC(ALM_AirAndWaterOK_T.DN)TON(H5b_On_T,?,?);
   48: [XIC(H5b_On_T.DN) XIO(GSC11) ,XIC(ALM_W1.26) XIO(AlarmReset) ]ADD(NumberOfAlarms,1,NumberOfAlarms)OTE(ALM_W1.26);
   // **************** Lower Hatch Failed to Raise and Lower Alarms ******************
   49: XIC(H4a)XIC(ALM_AirAndWaterOK_T.DN)TON(H4a_On_T,?,?);
   50: [XIC(H4a_On_T.DN) XIO(GSO10) ,XIC(ALM_W1.27) XIO(AlarmReset) ]ADD(NumberOfAlarms,1,NumberOfAlarms)OTE(ALM_W1.27);
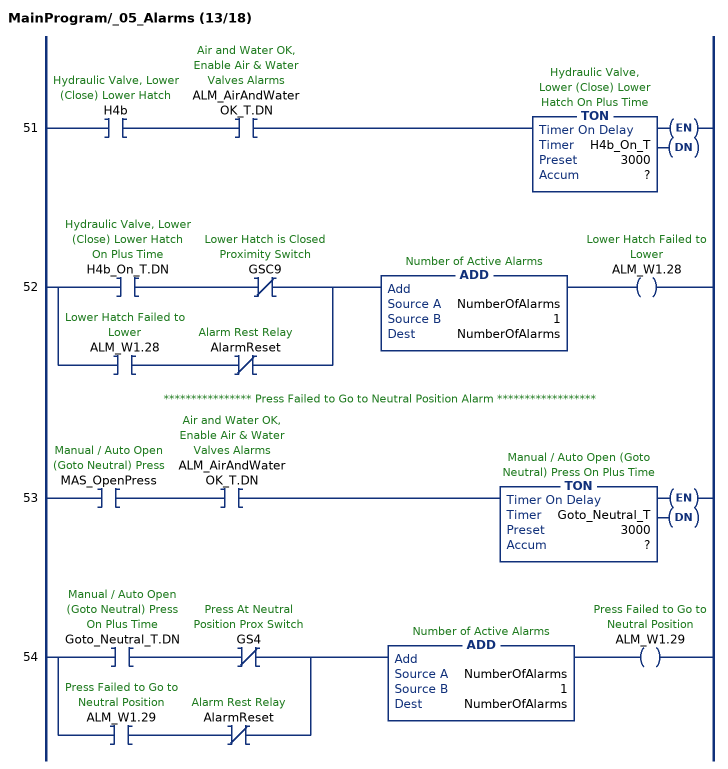
   51: XIC(H4b)XIC(ALM_AirAndWaterOK_T.DN)TON(H4b_On_T,?,?);
   52: [XIC(H4b_On_T.DN) XIO(GSC9) ,XIC(ALM_W1.28) XIO(AlarmReset) ]ADD(NumberOfAlarms,1,NumberOfAlarms)OTE(ALM_W1.28);
   // **************** Press Failed to Go to Neutral Position Alarm ******************
   53: XIC(MAS_OpenPress)XIC(ALM_AirAndWaterOK_T.DN)TON(Goto_Neutral_T,?,?);
   54: [XIC(Goto_Neutral_T.DN) XIO(GS4) ,XIC(ALM_W1.29) XIO(AlarmReset) ]ADD(NumberOfAlarms,1,NumberOfAlarms)OTE(ALM_W1.29);
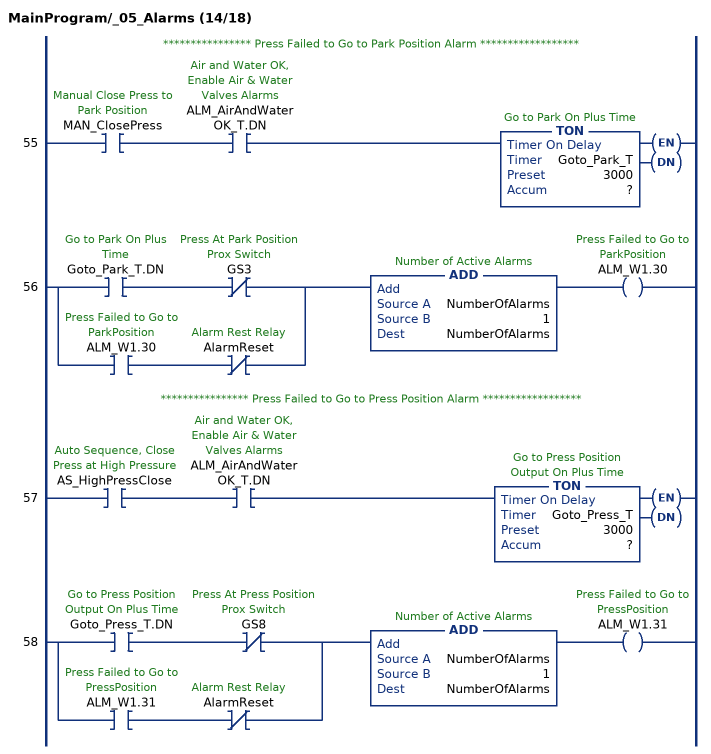
   // **************** Press Failed to Go to Park Position Alarm ******************
   55: XIC(MAN_ClosePress)XIC(ALM_AirAndWaterOK_T.DN)TON(Goto_Park_T,?,?);
   56: [XIC(Goto_Park_T.DN) XIO(GS3) ,XIC(ALM_W1.30) XIO(AlarmReset) ]ADD(NumberOfAlarms,1,NumberOfAlarms)OTE(ALM_W1.30);
   // **************** Press Failed to Go to Press Position Alarm ******************
   57: XIC(AS_HighPressClose)XIC(ALM_AirAndWaterOK_T.DN)TON(Goto_Press_T,?,?);
   58: [XIC(Goto_Press_T.DN) XIO(GS8) ,XIC(ALM_W1.31) XIO(AlarmReset) ]ADD(NumberOfAlarms,1,NumberOfAlarms)OTE(ALM_W1.31);
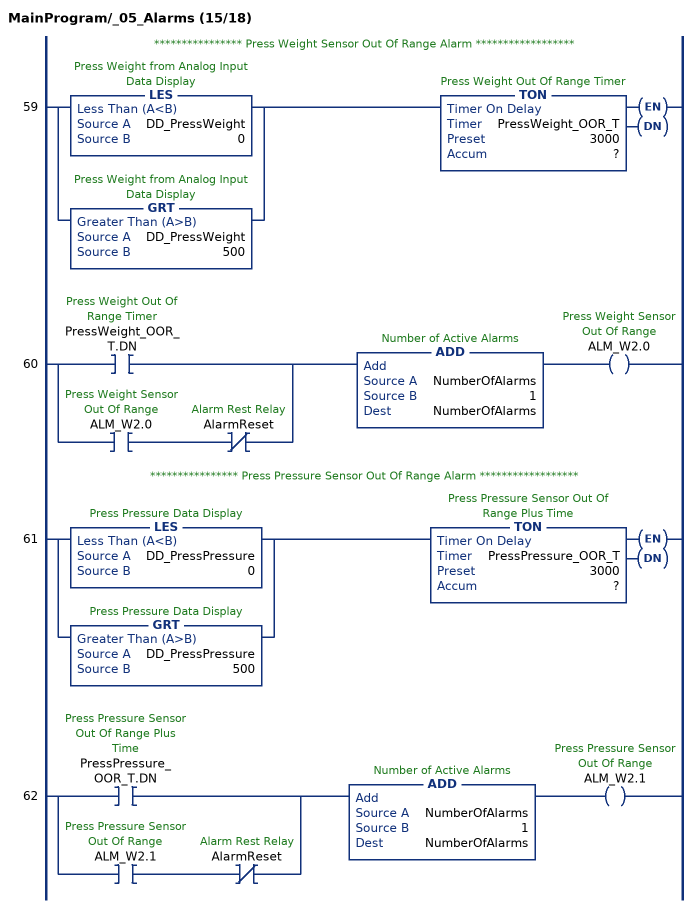
   // **************** Press Weight Sensor Out Of Range Alarm ******************
   59: [LES(DD_PressWeight,0) ,GRT(DD_PressWeight,500) ]TON(PressWeight_OOR_T,?,?);
   60: [XIC(PressWeight_OOR_T.DN) ,XIC(ALM_W2.0) XIO(AlarmReset) ]ADD(NumberOfAlarms,1,NumberOfAlarms)OTE(ALM_W2.0);
   // **************** Press Pressure Sensor Out Of Range Alarm ******************
   61: [LES(DD_PressPressure,0) ,GRT(DD_PressPressure,500) ]TON(PressPressure_OOR_T,?,?);
   62: [XIC(PressPressure_OOR_T.DN) ,XIC(ALM_W2.1) XIO(AlarmReset) ]ADD(NumberOfAlarms,1,NumberOfAlarms)OTE(ALM_W2.1);
